PROGRAM MAIN
VAR
	a : INT;
	b : INT;
	c : INT;
	
END_VAR

c := a+b;

END_PROGRAM

(* stored: Version 1.1.0.1, ProductVersion 3.1.4024.4
   POU MAIN: Id {56759815-ea35-437a-b440-8697e57be05b}, SpecialFunc None *)
